{attribute 'GeneratedUsingTerminal: EL9190--0000'}
{attribute addProperty BoxType "EL9190--0000"}
{attribute addProperty Description "EL9190 Power Supplier"}
{attribute addProperty Physics "KK"}
{attribute addProperty Id "EL9190"}
{attribute addProperty CRC "1494011728"}
{attribute addProperty Size "0"}
TYPE EL9190_590CCF50 EXTENDS EtcSlaveTerminalBase_947E5A46 :
STRUCT
END_STRUCT
END_TYPE

(* stored: Version 1.2.0.0, ProductVersion 3.1.4024.11
   DUT EL9190_590CCF50: Id {5cb3d699-5f17-4d52-96e5-c7cf988ea010} *)
